FUNCTION_BLOCK FB_Clock
VAR_INPUT
	bStartEnable : BOOL;
	fTimeStep : LREAL;
END_VAR
VAR_OUTPUT
	fTime : LREAL;
END_VAR
VAR
END_VAR


IF NOT(bStartEnable) THEN
	fTime := 0.0;
ELSE
	fTime := fTime + fTimeStep;
END_IF

END_FUNCTION_BLOCK

(* stored: Version 1.1.0.1
   POU FB_Clock: Id {b3566c58-5184-42a7-935d-777afebc62bf}, SpecialFunc None *)
